FUNCTION_BLOCK SimpleSort2Movers IMPLEMENTS I_DemoStep, I_BothMovers, I_Errorable
VAR_INPUT
		M1	:	I_XPlanarMover;
		M2	:	I_XPlanarMover;
END_VAR
VAR_OUTPUT
END_VAR
VAR
	_Done:BOOL;
	_Error: BOOL;
END_VAR

METHOD CyclicLogic
IF M1<>0 AND_THEN M2<>0 THEN
	_Error:=FALSE;
	IF M1.ActualPosition.y < M2.ActualPosition.y THEN
		ip.Movers[1] 	:= M1;
		ip.Movers[2] 	:= M2;	
	ELSE
		ip.Movers[2] 	:= M1;
		ip.Movers[1] 	:= M2;		
	END_IF	
	_Done:=TRUE;
ELSE
	_Error := TRUE;
END_IF
END_METHOD

{attribute 'monitoring' := 'call'}
PROPERTY Done : BOOL
GET
Done:=_Done;
END_GET
END_PROPERTY

PROPERTY Error : BOOL
GET
Error:= _Error;
END_GET
END_PROPERTY

PROPERTY Mover1 : I_XPlanarMover
GET
IF ip.Movers[1]<>0 THEN
	Mover1:=ip.Movers[1];
ELSE 
	Mover1:=M1;
END_IF
END_GET
SET
IF Mover1<>0 THEN
	ip.Movers[1]:=Mover1;
END_IF
END_SET
END_PROPERTY

PROPERTY Mover2 : I_XPlanarMover
GET
IF ip.Movers[2]<>0 THEN
	Mover2:=ip.Movers[2];
ELSE 
	Mover2:=M2;
END_IF
END_GET
SET
IF Mover2<>0 THEN
	ip.Movers[2]:=Mover2;
END_IF
END_SET
END_PROPERTY

METHOD Reset : BOOL
_Error:=FALSE;
_Done:=FALSE;
Reset:=TRUE;
END_METHOD

METHOD SetMovers : BOOL
VAR_INPUT
	M1	: I_XPlanarMover;
	M2	: I_XPlanarMover;
END_VAR
ip.Movers[1]:=M1;
ip.Movers[2]:=M2;
END_METHOD

END_FUNCTION_BLOCK

(* stored: Version 1.1.0.1, ProductVersion 3.1.4026.20
   POU SimpleSort2Movers: Id {0b3b5cc6-89d4-46ef-8516-83afbf2ef414}, SpecialFunc None
   Method CyclicLogic: Id {f4a31661-676b-45e8-a02a-ae3035f30584}
   Property Done: Id {18dbf2d2-ca2a-401a-b43f-85383008d1bc}
   Get Get: Id {0cec8e5e-cc21-41cb-85e5-3e493c0d6c2b}
   Property Error: Id {7b7382ba-c353-42de-96b6-03fa6bbcbec2}
   Get Get: Id {730bc7b3-caed-48a6-b2ee-9253c388e42a}
   Property Mover1: Id {d5b961fc-9c76-4767-ba35-2bfae814eefe}
   Get Get: Id {05b2b182-1aa5-4f5c-8c9d-2877cc22fd2f}
   Set Set: Id {48ed2f78-3450-48d3-8ab0-6c73b7bbc66b}
   Property Mover2: Id {47619d5a-00aa-4f9d-bac6-590d9ee7966c}
   Get Get: Id {ad920bf3-ba87-47b9-b518-ed5de68b6c40}
   Set Set: Id {91a5fc9a-25aa-4a1c-bcd8-bc8276ade7a5}
   Method Reset: Id {144e8ef9-aab5-42d7-8087-9dccb4daed16}
   Method SetMovers: Id {8903e4ff-9530-42a0-8b8f-0567619e0970} *)
